FUNCTION_BLOCK sequence_Pattern_08_08_loop_AX (* Pattern Sequence 8 Steps 8 Outputs (Cam Sequencer), AX Adapter *)
  (* Standard: 61499-2; Description: Copyright (c) 2026 HR Agrartechnik GmbH This program and the accompanying materials are made available under the terms of the Eclipse Public License 2.0 which is available at https://www.eclipse.org/legal/epl-2.0/ SPDX-License-Identifier: EPL-2.0 *)
  (* Version 1.0, 2026-02-01, Franz Höpfinger, HR Agrartechnik GmbH *)
  PACKAGE logiBUS::utils::sequence::pattern;
  IMPORT logiBUS::utils::sequence::const::sequence;
  IMPORT logiBUS::utils::sequence::const::sequence::NO_TIME;
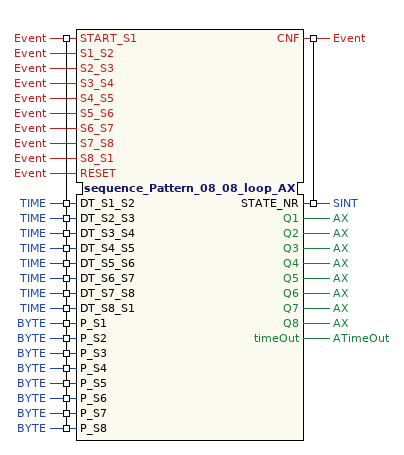
  EVENT_INPUT
    START_S1 WITH DT_S1_S2, DT_S2_S3, DT_S3_S4, DT_S4_S5, DT_S5_S6, DT_S6_S7, DT_S7_S8, DT_S8_S1, P_S1, P_S2, P_S3, P_S4, P_S5, P_S6, P_S7, P_S8; (* jump from START to State_01 *)
    S1_S2; (* jump from State_01 to State_02 *)
    S2_S3; (* jump from State_02 to State_03 *)
    S3_S4; (* jump from State_03 to State_04 *)
    S4_S5; (* jump from State_04 to State_05 *)
    S5_S6; (* jump from State_05 to State_06 *)
    S6_S7; (* jump from State_06 to State_07 *)
    S7_S8; (* jump from State_07 to State_08 *)
    S8_S1; (* jump from State_08 to State_01 *)
    RESET; (* Reset from any State to START *)
  END_EVENT
  EVENT_OUTPUT
    CNF WITH STATE_NR; (* Execution Confirmation *)
  END_EVENT
  VAR_INPUT
    DT_S1_S2 : TIME := NO_TIME; (* State_01 to State_02 timed *)
    DT_S2_S3 : TIME := NO_TIME; (* State_02 to State_03 timed *)
    DT_S3_S4 : TIME := NO_TIME; (* State_03 to State_04 timed *)
    DT_S4_S5 : TIME := NO_TIME; (* State_04 to State_05 timed *)
    DT_S5_S6 : TIME := NO_TIME; (* State_05 to State_06 timed *)
    DT_S6_S7 : TIME := NO_TIME; (* State_06 to State_07 timed *)
    DT_S7_S8 : TIME := NO_TIME; (* State_07 to State_08 timed *)
    DT_S8_S1 : TIME := NO_TIME; (* State_08 to State_01 timed *)
    P_S1 : BYTE := 1; (* Pattern for State 01 *)
    P_S2 : BYTE := 2; (* Pattern for State 02 *)
    P_S3 : BYTE := 4; (* Pattern for State 03 *)
    P_S4 : BYTE := 8; (* Pattern for State 04 *)
    P_S5 : BYTE := 16; (* Pattern for State 05 *)
    P_S6 : BYTE := 32; (* Pattern for State 06 *)
    P_S7 : BYTE := 64; (* Pattern for State 07 *)
    P_S8 : BYTE := 128; (* Pattern for State 08 *)
  END_VAR
  VAR_OUTPUT
    STATE_NR : SINT; (* State Number, START = 0, State_01 = 1... *)
  END_VAR
  PLUGS
    Q1 : adapter::types::unidirectional::AX; (* Output 1 (Bit 0) *)
    Q2 : adapter::types::unidirectional::AX; (* Output 2 (Bit 1) *)
    Q3 : adapter::types::unidirectional::AX; (* Output 3 (Bit 2) *)
    Q4 : adapter::types::unidirectional::AX; (* Output 4 (Bit 3) *)
    Q5 : adapter::types::unidirectional::AX; (* Output 5 (Bit 4) *)
    Q6 : adapter::types::unidirectional::AX; (* Output 6 (Bit 5) *)
    Q7 : adapter::types::unidirectional::AX; (* Output 7 (Bit 6) *)
    Q8 : adapter::types::unidirectional::AX; (* Output 8 (Bit 7) *)
    timeOut : iec61499::events::ATimeOut; (* timeOut Adapter *)
  END_PLUGS
  EC_STATES
    xSTART; (* Initial State *)
    sState_01 : -> timeOut.STOP, State_01_C -> CNF, State_01_E -> Q1.E1, -> Q2.E1, -> Q3.E1, -> Q4.E1, -> Q5.E1, -> Q6.E1, -> Q7.E1, -> Q8.E1, -> timeOut.START;
    sState_02 : -> timeOut.STOP, State_02_C -> CNF, State_02_E -> Q1.E1, -> Q2.E1, -> Q3.E1, -> Q4.E1, -> Q5.E1, -> Q6.E1, -> Q7.E1, -> Q8.E1, -> timeOut.START;
    sState_03 : -> timeOut.STOP, State_03_C -> CNF, State_03_E -> Q1.E1, -> Q2.E1, -> Q3.E1, -> Q4.E1, -> Q5.E1, -> Q6.E1, -> Q7.E1, -> Q8.E1, -> timeOut.START;
    sState_04 : -> timeOut.STOP, State_04_C -> CNF, State_04_E -> Q1.E1, -> Q2.E1, -> Q3.E1, -> Q4.E1, -> Q5.E1, -> Q6.E1, -> Q7.E1, -> Q8.E1, -> timeOut.START;
    sState_05 : -> timeOut.STOP, State_05_C -> CNF, State_05_E -> Q1.E1, -> Q2.E1, -> Q3.E1, -> Q4.E1, -> Q5.E1, -> Q6.E1, -> Q7.E1, -> Q8.E1, -> timeOut.START;
    sState_06 : -> timeOut.STOP, State_06_C -> CNF, State_06_E -> Q1.E1, -> Q2.E1, -> Q3.E1, -> Q4.E1, -> Q5.E1, -> Q6.E1, -> Q7.E1, -> Q8.E1, -> timeOut.START;
    sState_07 : -> timeOut.STOP, State_07_C -> CNF, State_07_E -> Q1.E1, -> Q2.E1, -> Q3.E1, -> Q4.E1, -> Q5.E1, -> Q6.E1, -> Q7.E1, -> Q8.E1, -> timeOut.START;
    sState_08 : -> timeOut.STOP, State_08_C -> CNF, State_08_E -> Q1.E1, -> Q2.E1, -> Q3.E1, -> Q4.E1, -> Q5.E1, -> Q6.E1, -> Q7.E1, -> Q8.E1, -> timeOut.START;
    sRESET : -> timeOut.STOP, RESET_Outs -> Q1.E1, -> Q2.E1, -> Q3.E1, -> Q4.E1, -> Q5.E1, -> Q6.E1, -> Q7.E1, -> Q8.E1, State_00_C -> CNF;
  END_STATES
  EC_TRANSITIONS
    sState_01 TO sState_02 := S1_S2;
    sState_02 TO sState_03 := S2_S3;
    sState_03 TO sState_04 := S3_S4;
    sState_04 TO sState_05 := S4_S5;
    sState_05 TO sState_06 := S5_S6;
    sState_06 TO sState_07 := S6_S7;
    sState_07 TO sState_08 := S7_S8;
    sState_08 TO sState_01 := S8_S1;
    sState_01 TO sState_02 := timeOut.TimeOut;
    sState_02 TO sState_03 := timeOut.TimeOut;
    sState_03 TO sState_04 := timeOut.TimeOut;
    sState_04 TO sState_05 := timeOut.TimeOut;
    sState_05 TO sState_06 := timeOut.TimeOut;
    sState_06 TO sState_07 := timeOut.TimeOut;
    sState_07 TO sState_08 := timeOut.TimeOut;
    sState_08 TO sState_01 := timeOut.TimeOut;
    xSTART TO sState_01 := START_S1;
    sState_01 TO sRESET := RESET;
    sState_02 TO sRESET := RESET;
    sState_03 TO sRESET := RESET;
    sState_04 TO sRESET := RESET;
    sState_05 TO sRESET := RESET;
    sState_06 TO sRESET := RESET;
    sState_07 TO sRESET := RESET;
    sState_08 TO sRESET := RESET;
    sRESET TO xSTART := 1;
  END_TRANSITIONS
  ALGORITHM State_00_C IN ST:
STATE_NR := sequence::State_00;
  END_ALGORITHM
  ALGORITHM State_01_C IN ST:
STATE_NR := sequence::State_01;
timeOut.DT := DT_S1_S2;
  END_ALGORITHM
  ALGORITHM State_02_C IN ST:
STATE_NR := sequence::State_02;
timeOut.DT := DT_S2_S3;
  END_ALGORITHM
  ALGORITHM State_03_C IN ST:
STATE_NR := sequence::State_03;
timeOut.DT := DT_S3_S4;
  END_ALGORITHM
  ALGORITHM State_04_C IN ST:
STATE_NR := sequence::State_04;
timeOut.DT := DT_S4_S5;
  END_ALGORITHM
  ALGORITHM State_05_C IN ST:
STATE_NR := sequence::State_05;
timeOut.DT := DT_S5_S6;
  END_ALGORITHM
  ALGORITHM State_06_C IN ST:
STATE_NR := sequence::State_06;
timeOut.DT := DT_S6_S7;
  END_ALGORITHM
  ALGORITHM State_07_C IN ST:
STATE_NR := sequence::State_07;
timeOut.DT := DT_S7_S8;
  END_ALGORITHM
  ALGORITHM State_08_C IN ST:
STATE_NR := sequence::State_08;
timeOut.DT := DT_S8_S1;
  END_ALGORITHM
  ALGORITHM State_01_E IN ST:
Q1.D1 := P_S1.0;
Q2.D1 := P_S1.1;
Q3.D1 := P_S1.2;
Q4.D1 := P_S1.3;
Q5.D1 := P_S1.4;
Q6.D1 := P_S1.5;
Q7.D1 := P_S1.6;
Q8.D1 := P_S1.7;
  END_ALGORITHM
  ALGORITHM State_02_E IN ST:
Q1.D1 := P_S2.0;
Q2.D1 := P_S2.1;
Q3.D1 := P_S2.2;
Q4.D1 := P_S2.3;
Q5.D1 := P_S2.4;
Q6.D1 := P_S2.5;
Q7.D1 := P_S2.6;
Q8.D1 := P_S2.7;
  END_ALGORITHM
  ALGORITHM State_03_E IN ST:
Q1.D1 := P_S3.0;
Q2.D1 := P_S3.1;
Q3.D1 := P_S3.2;
Q4.D1 := P_S3.3;
Q5.D1 := P_S3.4;
Q6.D1 := P_S3.5;
Q7.D1 := P_S3.6;
Q8.D1 := P_S3.7;
  END_ALGORITHM
  ALGORITHM State_04_E IN ST:
Q1.D1 := P_S4.0;
Q2.D1 := P_S4.1;
Q3.D1 := P_S4.2;
Q4.D1 := P_S4.3;
Q5.D1 := P_S4.4;
Q6.D1 := P_S4.5;
Q7.D1 := P_S4.6;
Q8.D1 := P_S4.7;
  END_ALGORITHM
  ALGORITHM State_05_E IN ST:
Q1.D1 := P_S5.0;
Q2.D1 := P_S5.1;
Q3.D1 := P_S5.2;
Q4.D1 := P_S5.3;
Q5.D1 := P_S5.4;
Q6.D1 := P_S5.5;
Q7.D1 := P_S5.6;
Q8.D1 := P_S5.7;
  END_ALGORITHM
  ALGORITHM State_06_E IN ST:
Q1.D1 := P_S6.0;
Q2.D1 := P_S6.1;
Q3.D1 := P_S6.2;
Q4.D1 := P_S6.3;
Q5.D1 := P_S6.4;
Q6.D1 := P_S6.5;
Q7.D1 := P_S6.6;
Q8.D1 := P_S6.7;
  END_ALGORITHM
  ALGORITHM State_07_E IN ST:
Q1.D1 := P_S7.0;
Q2.D1 := P_S7.1;
Q3.D1 := P_S7.2;
Q4.D1 := P_S7.3;
Q5.D1 := P_S7.4;
Q6.D1 := P_S7.5;
Q7.D1 := P_S7.6;
Q8.D1 := P_S7.7;
  END_ALGORITHM
  ALGORITHM State_08_E IN ST:
Q1.D1 := P_S8.0;
Q2.D1 := P_S8.1;
Q3.D1 := P_S8.2;
Q4.D1 := P_S8.3;
Q5.D1 := P_S8.4;
Q6.D1 := P_S8.5;
Q7.D1 := P_S8.6;
Q8.D1 := P_S8.7;
  END_ALGORITHM
  ALGORITHM RESET_Outs IN ST:
Q1.D1 := FALSE;
Q2.D1 := FALSE;
Q3.D1 := FALSE;
Q4.D1 := FALSE;
Q5.D1 := FALSE;
Q6.D1 := FALSE;
Q7.D1 := FALSE;
Q8.D1 := FALSE;
  END_ALGORITHM
END_FUNCTION_BLOCK
